Staubli VAL3: start.pgx

public program start()
  local num i
  local num l_nKey
  local string l_sMessage
begin
  // call the start
  taskCreate "KERNEL",100,kernel:start()
end
